KUKA KRL data list: LAB_NATIVE.dat

&ACCESS RVP
&REL 1
DEFDAT LAB_NATIVE PUBLIC
ENDDAT
